// TIA Portal V20 export
// export: Created 2026-07-10T11:12:35.1642312Z, ExportSetting WithDefaults, DisplayName Totally Integrated Automation Portal, DisplayVersion V20, DisplayName TIA Portal Openness, DisplayVersion V20, DisplayName TIA Portal Version Control Interface, DisplayVersion V20, DisplayName STEP 7 Professional, DisplayVersion V20, DisplayName STEP 7 Safety, DisplayVersion V20, DisplayName WinCC Basic/Comfort/Advanced, DisplayVersion V20, DisplayName WinCC Unified, DisplayVersion V20
FUNCTION_BLOCK "ChlorConsumptionAlarm"   // FB6, SCL
{ S7_Optimized_Access := 'TRUE' }
VERSION : 0.1
// stored: AutoNumber true, IsIECCheckEnabled false, IsRetainMemResEnabled false, MemoryReserve 100, SetENOAutomatically false, UDAEnableTagReadback false
   VAR_OUTPUT
      HighAlarm : Bool;
   END_VAR
   VAR
      "step" : Int;
      maxConsamption : Real;
      monitorTime : Real;
      weightNow : Real;
      weightLast : Real;
      TON { S7_SetPoint := 'True'} : TON_TIME;
      weightDelta { S7_SetPoint := 'True'} : Real;
   END_VAR
BEGIN
   #maxConsamption := "MB".Table.ChlorConsumptionTable[0].Consumption;
   #monitorTime := "MB".Table.ChlorConsumptionTable[0].MonitorTIme;

   IF "MB".Table.CycleDay >= "MB".Table.ChlorConsumptionTable[3].Day THEN
       #maxConsamption := "MB".Table.ChlorConsumptionTable[3].Consumption;
       #monitorTime    := "MB".Table.ChlorConsumptionTable[3].MonitorTIme;
   ELSIF "MB".Table.CycleDay >= "MB".Table.ChlorConsumptionTable[2].Day THEN
       #maxConsamption := "MB".Table.ChlorConsumptionTable[2].Consumption;
       #monitorTime    := "MB".Table.ChlorConsumptionTable[2].MonitorTIme;
   ELSIF "MB".Table.CycleDay >= "MB".Table.ChlorConsumptionTable[1].Day THEN
       #maxConsamption := "MB".Table.ChlorConsumptionTable[1].Consumption;
       #monitorTime    := "MB".Table.ChlorConsumptionTable[1].MonitorTIme;
   ELSIF "MB".Table.CycleDay >= "MB".Table.ChlorConsumptionTable[0].Day THEN
       #maxConsamption := "MB".Table.ChlorConsumptionTable[0].Consumption;
       #monitorTime    := "MB".Table.ChlorConsumptionTable[0].MonitorTIme;
   END_IF;

   #TON(IN:=TRUE,
        PT:=REAL_TO_DINT(#monitorTime*3600*1000));

   IF #TON.Q THEN
       #weightLast := #weightNow;
       RESET_TIMER(#TON);
   END_IF;
   #weightNow := "MB".Table.WeightValue1Liters;
   #weightDelta := #weightLast - #weightNow;


   IF "MB".Table.HMI_WeightAlarmReset THEN
       #weightDelta := 0;
       #weightNow := "MB".Table.WeightValue1Liters;
       #weightLast := #weightNow;
       #HighAlarm := false;
       RESET_TIMER(#TON);
       "MB".Table.HMI_WeightAlarmReset := FALSE;
   END_IF;

   IF #weightDelta > #maxConsamption THEN
       #HighAlarm := TRUE;
   END_IF;
END_FUNCTION_BLOCK
